INTERFACE itfCommand

METHOD Abort : MC_Error
END_METHOD

PROPERTY Active : BOOL
GET
END_GET
END_PROPERTY

PROPERTY Busy : BOOL
GET
END_GET
END_PROPERTY

PROPERTY Command : MC_COMMAND_REF
GET
END_GET
END_PROPERTY

PROPERTY CommandAborted : BOOL
GET
END_GET
END_PROPERTY

PROPERTY Done : BOOL
GET
END_GET
END_PROPERTY

PROPERTY Error : BOOL
GET
END_GET
END_PROPERTY

PROPERTY ErrorId : MC_Error
GET
END_GET
END_PROPERTY

METHOD Wait : MC_Error
VAR_INPUT
	Timeout: TIME;
	AbortOnTimeout: BOOL;
END_VAR
END_METHOD

END_INTERFACE

(* stored: Version 1.1.0.1, ProductVersion 3.1.4024.11
   Itf itfCommand: Id {808308aa-5be1-474f-9cd7-f693a8f9904a}
   Method Abort: Id {8b5e35ac-b5b0-4aa3-ac23-dd574710cbdb}
   Property Active: Id {ee573e9a-5ea0-49eb-8a77-58c3db89cb06}
   Get Get: Id {e352ae0e-c36b-4b81-925e-c16793043b20}
   Property Busy: Id {219c6516-004b-45fc-b650-7ed67eb9c5f4}
   Get Get: Id {70a9e6f3-edce-4f63-b2c1-423f4fda519b}
   Property Command: Id {75a96964-1bda-4b50-a0bc-30c1d7adea11}
   Get Get: Id {8be75cdb-2b18-48a1-bc6a-42a770e708c0}
   Property CommandAborted: Id {1228aed1-e6c8-4a0c-83a8-614a39b5cd17}
   Get Get: Id {fb1159f9-2f74-4c35-9b7c-b8e426978d69}
   Property Done: Id {d40ac11d-8d91-4f20-b524-e82b3a89ff64}
   Get Get: Id {68784eb7-567c-47e4-8ee8-ee6c175661f0}
   Property Error: Id {3c0e0fa2-bc73-41b1-b093-306901cd5baf}
   Get Get: Id {da0594a0-bb9a-4f73-88c6-5ba58a46ceea}
   Property ErrorId: Id {fef3784f-c132-4b1e-9f11-d65718464c45}
   Get Get: Id {88815e75-2241-4565-8dad-370d99d2e3d8}
   Method Wait: Id {14133628-3c21-4d21-a48c-496a1b395288} *)
